FUNCTION_BLOCK Mc3StopTask EXTENDS Mc3MotionTask IMPLEMENTS I_Mc3MotionTask
VAR
	McHalt : Tc3_Mc3Ptp.MC_Halt;
END_VAR

{attribute 'monitoring' := 'call'}
PROPERTY Busy : BOOL
GET
Busy := McHalt.Busy;
END_GET
END_PROPERTY

METHOD CyclicLogic
McHalt(Axis			  := _Axis.Axis,
	   Deceleration	  := _Axis.Deceleration,
	   Jerk			  := _Axis.Jerk,
	   Done			  =>,
	   Busy			  =>,
	   Active		  =>,
	   CommandAborted =>,
	   Error		  =>,
	   ErrorId		  =>);

McHalt.Execute := FALSE;
END_METHOD

{attribute 'monitoring' := 'call'}
PROPERTY Error : BOOL
GET
Error := McHalt.Error;
END_GET
END_PROPERTY

{attribute 'monitoring' := 'call'}
PROPERTY ErrorId : UDINT
GET
ErrorId := McHalt.ErrorID;
END_GET
END_PROPERTY

METHOD Execute : BOOL
McHalt(Axis			:= _Axis.Axis,
	   Execute		:= TRUE,
	   Deceleration := _Axis.Deceleration,
	   Jerk			:= _Axis.Jerk);

Execute := TRUE;
END_METHOD

END_FUNCTION_BLOCK

(* stored: Version 1.1.0.1, ProductVersion 3.1.4026.20
   POU Mc3StopTask: Id {d77fbe87-6105-464c-9436-a66cec7c7ae4}, SpecialFunc None
   Property Busy: Id {a4d84e5c-eaba-4869-8701-28bac64cc300}
   Get Get: Id {9d27e6ef-8c3c-4ebf-82b7-773d6240a069}
   Method CyclicLogic: Id {c3e780ea-a070-4cf4-b6da-5aef2c425231}
   Property Error: Id {7bd9da7b-7384-4b09-9be8-e5c1e5b31669}
   Get Get: Id {9acc4f28-6d6b-43f1-b85e-aa81549dc3f4}
   Property ErrorId: Id {44e53075-5f67-4ffb-a2d7-f77d2823e989}
   Get Get: Id {dcd257a6-ad9d-4683-a829-13f2c33d098d}
   Method Execute: Id {4e7ea144-6046-4cf7-80d9-8af8a6a3f982} *)
